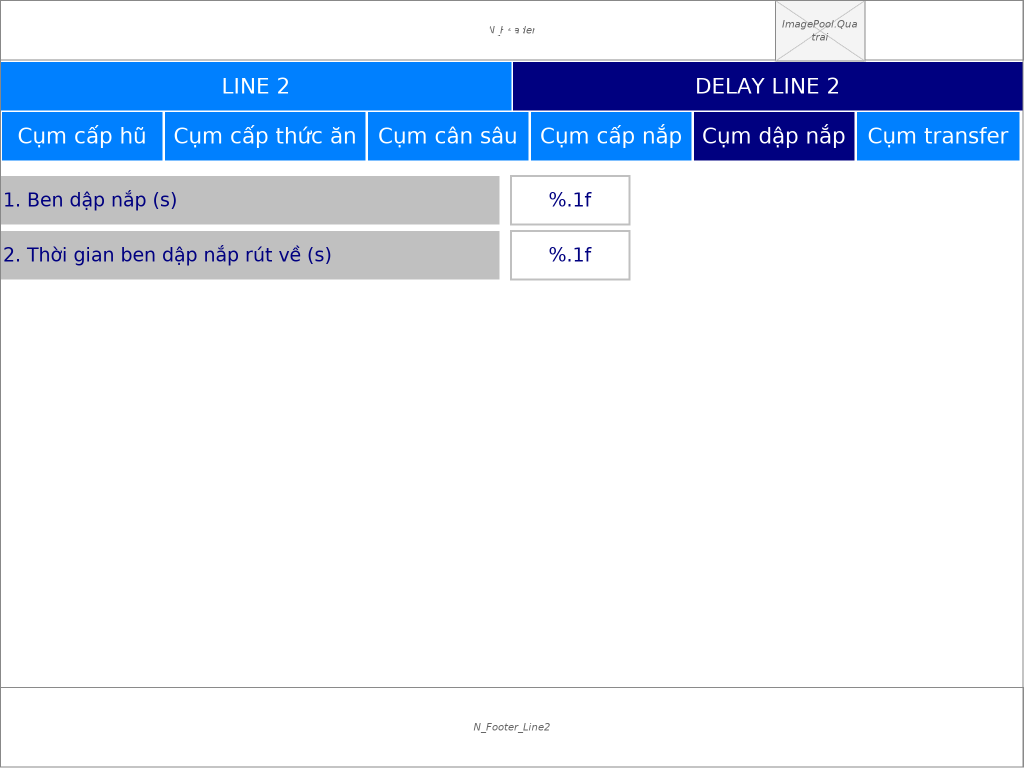
VISUALIZATION N_Setting_Delay_LidPressing2  // 1024x768
    Frame (0,687 1024x80)
        shows N_Footer_Line2()
    Frame (0,0 1024x60)
        shows N_Header()
    Textfield (353,4 420x50), "MÀN HÌNH CÀI KHOẢNG TRỄ LINE 2"
    Rectangle (0,175 500x50), "1. Ben dập nắp (s)"
    Rectangle (0,230 500x50), "2. Thời gian ben dập nắp rút về (s)"
    Rectangle (0,61 512x50), "LINE 2"
        OnMouseClick: change screen: N_Setting_Line2
    Rectangle (1,111 162x50), "Cụm cấp hũ"
        OnMouseClick: change screen: N_Setting_Delay_JarSupply2
    Rectangle (164,111 202x50), "Cụm cấp thức ăn"
        OnMouseClick: change screen: N_Setting_Delay_FoodSupply2
    Rectangle (367,111 162x50), "Cụm cân sâu"
        OnMouseClick: change screen: N_Setting_Delay_WorwWeight2
    Rectangle (530,111 162x50), "Cụm cấp nắp"
        OnMouseClick: change screen: N_Setting_Delay_LidSupply2
    Rectangle (693,111 162x50), "Cụm dập nắp"
        OnMouseClick: change screen: N_Setting_Delay_LidPressing2
    Rectangle (856,111 164x50), "Cụm transfer"
        OnMouseClick: change screen: N_Setting_Delay_Tranfer2
    Rectangle (512,61 511x50), "DELAY LINE 2"
        OnMouseClick: change screen: N_Setting_Delay_JarSupply2
    Image (775,0 90x61), image: ImagePool.Qua trai
        OnMouseClick: change screen: N_Setting_Delay_LidPressing1
    Rectangle (510,175 120x50), "%.1f", text variable: PR_Line02.timer_Check_Cylinder_extend
        OnMouseClick: write PR_Line02.timer_Check_Cylinder_extend via VisuDialogs.Numpad
    Rectangle (510,230 120x50), "%.1f", text variable: PR_Line02.timer_Check_Cylinder_retract
        OnMouseClick: write PR_Line02.timer_Check_Cylinder_retract via VisuDialogs.Numpad
END_VISUALIZATION

(* stored: Version 1.1.0.1, ProductVersion 3.1.4024.12
   Visu N_Setting_Delay_LidPressing2: Id {63228fb5-c60f-4080-a556-3e7f74c16d91} *)
